// TIA Portal project "Carroponte" (V16)

(* hardware
DEVICE "S7-1200 station_1"  S7-1200 Station
   slot 0: "Telaio di montaggio_0"  S7-1200 Rack  Rack  V1.0
   slot 1: "PLC_1"  CPU 1214C DC/DC/DC  6ES7 214-1AG40-0XB0  V4.1
*)

// ===== PLC "PLC_1"  CPU 1214C DC/DC/DC =====

VAR_GLOBAL   // PLC tag table "Tabella delle variabili standard"
   "START" AT %I0.0 : Bool;
   "SDown" AT %I0.1 : Bool;
   "SUp" AT %I0.2 : Bool;
   "S1" AT %I0.3 : Bool;
   "S2" AT %I0.4 : Bool;
   "Left" AT %Q0.0 : Bool;
   "Right" AT %Q0.1 : Bool;
   "Down" AT %Q0.2 : Bool;
   "Up" AT %Q0.3 : Bool;
   "S3" AT %I0.5 : Bool;
END_VAR

VAR_GLOBAL CONSTANT   // PLC tag table "Tabella delle variabili standard"
   "TEMPO_TRASCORSO" : Time := T#15s;
END_VAR

DATA_BLOCK "VariabiliDiStato"   // DB1
{ S7_Optimized_Access := 'TRUE' }
VERSION : 0.1
   VAR RETAIN
      HOME : Bool := true;
      Destra1 : Bool;
      Su : Bool;
      Destra2 : Bool;
      Attesa : Bool;
      Sinistra : Bool;
      Giù : Bool;
   END_VAR
BEGIN
END_DATA_BLOCK

// folder: System blocks/Program resources

DATA_BLOCK "IEC_Timer_0_DB"   // DB2
{ S7_Optimized_Access := 'TRUE' }
AUTHOR : Simatic
FAMILY : IEC
NAME : IEC_TMR
VERSION : 1.0
// stored: InstanceOfName IEC_TIMER
"IEC_TIMER"
BEGIN
END_DATA_BLOCK

// folder: (top level)

ORGANIZATION_BLOCK "Main"   // OB1, LAD, ProgramCycle
TITLE = "Main Program Sweep (Cycle)"
{ S7_Optimized_Access := 'TRUE' }
VERSION : 0.1
   VAR_INPUT
      Initial_Call : Bool;   // Initial call of this OB
      Remanence : Bool;   // =True, if remanent data are available
   END_VAR
BEGIN

REGION Network 1
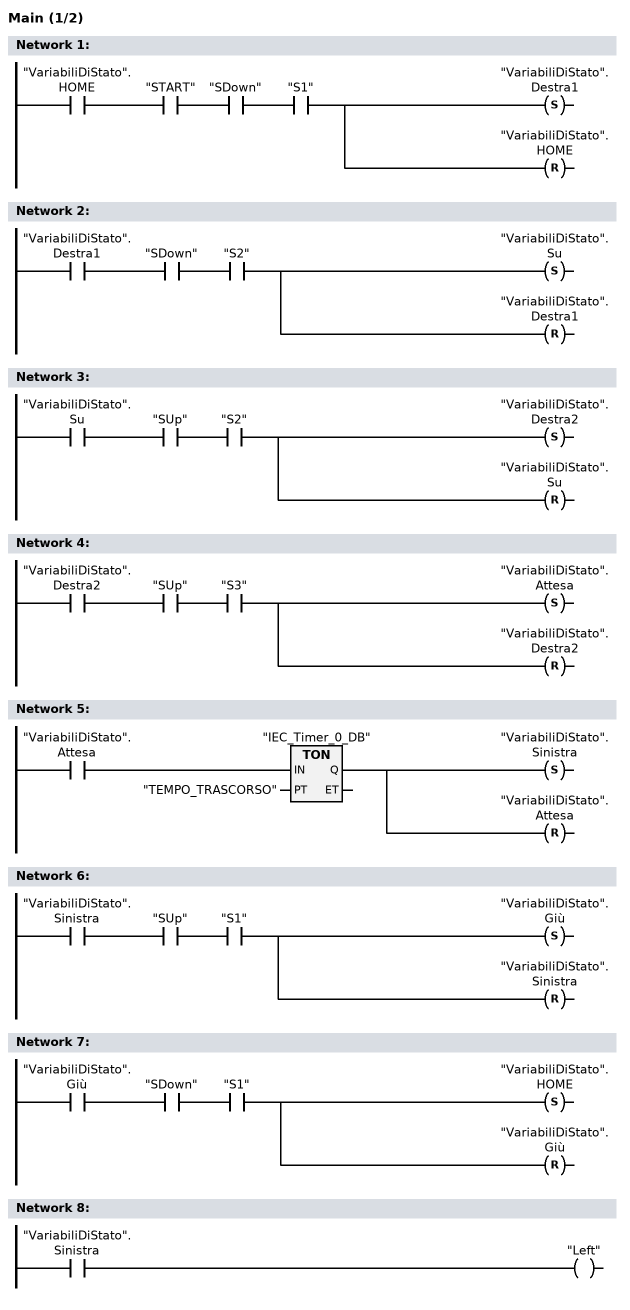
   RUNG wire#powerrail
      Contact( "VariabiliDiStato".HOME )
      Contact( "START" )
      Contact( "SDown" )
      Contact( "S1" )
      wire#w1
      S_Coil( "VariabiliDiStato".Destra1 )
   END_RUNG
   RUNG wire#w1
      R_Coil( "VariabiliDiStato".HOME )
   END_RUNG
   // the same network as SCL:
   IF "VariabiliDiStato".HOME AND "START" AND "SDown" AND "S1" THEN
       "VariabiliDiStato".Destra1 := TRUE;
       "VariabiliDiStato".HOME := FALSE;
   END_IF;
END_REGION

REGION Network 2
   RUNG wire#powerrail
      Contact( "VariabiliDiStato".Destra1 )
      Contact( "SDown" )
      Contact( "S2" )
      wire#w1
      S_Coil( "VariabiliDiStato".Su )
   END_RUNG
   RUNG wire#w1
      R_Coil( "VariabiliDiStato".Destra1 )
   END_RUNG
   // the same network as SCL:
   IF "VariabiliDiStato".Destra1 AND "SDown" AND "S2" THEN
       "VariabiliDiStato".Su := TRUE;
       "VariabiliDiStato".Destra1 := FALSE;
   END_IF;
END_REGION

REGION Network 3
   RUNG wire#powerrail
      Contact( "VariabiliDiStato".Su )
      Contact( "SUp" )
      Contact( "S2" )
      wire#w1
      S_Coil( "VariabiliDiStato".Destra2 )
   END_RUNG
   RUNG wire#w1
      R_Coil( "VariabiliDiStato".Su )
   END_RUNG
   // the same network as SCL:
   IF "VariabiliDiStato".Su AND "SUp" AND "S2" THEN
       "VariabiliDiStato".Destra2 := TRUE;
       "VariabiliDiStato".Su := FALSE;
   END_IF;
END_REGION

REGION Network 4
   RUNG wire#powerrail
      Contact( "VariabiliDiStato".Destra2 )
      Contact( "SUp" )
      Contact( "S3" )
      wire#w1
      S_Coil( "VariabiliDiStato".Attesa )
   END_RUNG
   RUNG wire#w1
      R_Coil( "VariabiliDiStato".Destra2 )
   END_RUNG
   // the same network as SCL:
   IF "VariabiliDiStato".Destra2 AND "SUp" AND "S3" THEN
       "VariabiliDiStato".Attesa := TRUE;
       "VariabiliDiStato".Destra2 := FALSE;
   END_IF;
END_REGION

REGION Network 5
   "IEC_Timer_0_DB".TON(IN := "VariabiliDiStato".Attesa, PT := "TEMPO_TRASCORSO");
   IF "IEC_Timer_0_DB".Q THEN
       "VariabiliDiStato".Sinistra := TRUE;
       "VariabiliDiStato".Attesa := FALSE;
   END_IF;
END_REGION

REGION Network 6
   RUNG wire#powerrail
      Contact( "VariabiliDiStato".Sinistra )
      Contact( "SUp" )
      Contact( "S1" )
      wire#w1
      S_Coil( "VariabiliDiStato".Giù )
   END_RUNG
   RUNG wire#w1
      R_Coil( "VariabiliDiStato".Sinistra )
   END_RUNG
   // the same network as SCL:
   IF "VariabiliDiStato".Sinistra AND "SUp" AND "S1" THEN
       "VariabiliDiStato".Giù := TRUE;
       "VariabiliDiStato".Sinistra := FALSE;
   END_IF;
END_REGION

REGION Network 7
   RUNG wire#powerrail
      Contact( "VariabiliDiStato".Giù )
      Contact( "SDown" )
      Contact( "S1" )
      wire#w1
      S_Coil( "VariabiliDiStato".HOME )
   END_RUNG
   RUNG wire#w1
      R_Coil( "VariabiliDiStato".Giù )
   END_RUNG
   // the same network as SCL:
   IF "VariabiliDiStato".Giù AND "SDown" AND "S1" THEN
       "VariabiliDiStato".HOME := TRUE;
       "VariabiliDiStato".Giù := FALSE;
   END_IF;
END_REGION

REGION Network 8
   RUNG wire#powerrail
      Contact( "VariabiliDiStato".Sinistra )
      Coil( "Left" )
   END_RUNG
   // the same network as SCL:
   "Left" := "VariabiliDiStato".Sinistra;
END_REGION

REGION Network 9
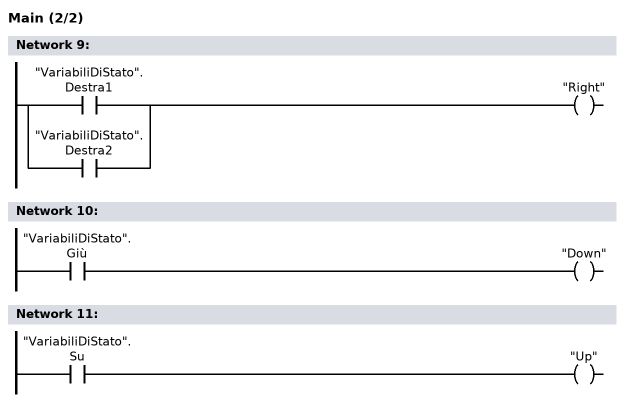
   RUNG wire#powerrail
      Contact( "VariabiliDiStato".Destra1 )
      wire#w1
      Coil( "Right" )
   END_RUNG
   RUNG wire#powerrail
      Contact( "VariabiliDiStato".Destra2 )
   END_RUNG wire#w1
   // the same network as SCL:
   "Right" := "VariabiliDiStato".Destra1 OR "VariabiliDiStato".Destra2;
END_REGION

REGION Network 10
   RUNG wire#powerrail
      Contact( "VariabiliDiStato".Giù )
      Coil( "Down" )
   END_RUNG
   // the same network as SCL:
   "Down" := "VariabiliDiStato".Giù;
END_REGION

REGION Network 11
   RUNG wire#powerrail
      Contact( "VariabiliDiStato".Su )
      Coil( "Up" )
   END_RUNG
   // the same network as SCL:
   "Up" := "VariabiliDiStato".Su;
END_REGION
END_ORGANIZATION_BLOCK